FUNCTION_BLOCK ABSTRACT FB_Collections IMPLEMENTS I_Collections
VAR
	stError : ST_ERROR;
	nCount 	: DINT; // Size of Collection
END_VAR

(* Number of items in the collection *)
PROPERTY _Count : DINT
GET
_Count := THIS^.nCount;
END_GET
END_PROPERTY

(* Gets collection's error status *)
PROPERTY _Error_Status : ST_ERROR
GET
_Error_Status := THIS^.stError;
END_GET
END_PROPERTY

(* Checks if collection is empty.*)
PROPERTY _Is_Empty : BOOL
GET
END_GET
END_PROPERTY

(* Empties/Clears/Deletes every element on the collection*)
METHOD Clear
END_METHOD

END_FUNCTION_BLOCK

(* stored: Version 1.1.0.1, ProductVersion 3.1.4024.4
   POU FB_Collections: Id {7e0153eb-1d71-478f-9767-a8d202b4be94}, SpecialFunc None
   Property _Count: Id {78d04743-c673-4006-9846-92d78266d4b2}
   Get Get: Id {ae399a3c-7dcf-43a1-8adb-3a201539dc8f}
   Property _Error_Status: Id {f5c500f3-5fca-40ca-920d-3a5de241efb2}
   Get Get: Id {fd22dab7-ee66-4cce-994c-2910fa8e58fb}
   Property _Is_Empty: Id {bda19a5b-6eae-4b14-8f4f-ed4cf062299f}
   Get Get: Id {bdf3428d-3c6e-416d-9454-b5bf770d84a5}
   Method Clear: Id {0584369c-c17b-4cbe-8e4d-6d1d31ac2e96} *)
